PROGRAM SYSTEM
VAR
	fbGetCurTaskIdx  : GETCURTASKINDEX; // PlcTaskSystemInfo for Cycle time
	
	
END_VAR

fbGetCurTaskIdx();
GVL.CycleTime := _TaskInfo[fbGetCurTaskIdx.index].CycleTime/10000;

GVL.GetLocalSystemTimeFB(
	sNetID:= , 
	bEnable:= TRUE, 
	dwCycle:= 1, 
	dwOpt:= , 
	tTimeout:= , 
	bValid=> , 
	systemTime=> , 
	tzID=> );
	
GVL.SystemDateTime := SYSTEMTIME_TO_STRING(GVL.GetLocalSystemTimeFB.systemTime);

GVL.SystemDate := MID(STR:=GVL.SystemDateTime , LEN:=10 , POS:=1 );
GVL.SystemTime := MID(STR:=GVL.SystemDateTime , LEN:=8 , POS:=12 );

END_PROGRAM

(* stored: Version 1.1.0.1, ProductVersion 3.1.4024.12
   POU SYSTEM: Id {8a0e2ec5-91f0-4231-a4cd-9f6327880700}, SpecialFunc None *)
